// TIA Portal V19 export
FUNCTION "BACKWASH" : Void   // FC13, LAD
{ S7_Optimized_Access := 'TRUE' }
// stored: SetENOAutomatically false
BEGIN

REGION Network 1: BACKWASH_TIMER
END_REGION

REGION Network 2: VALVE OPEN
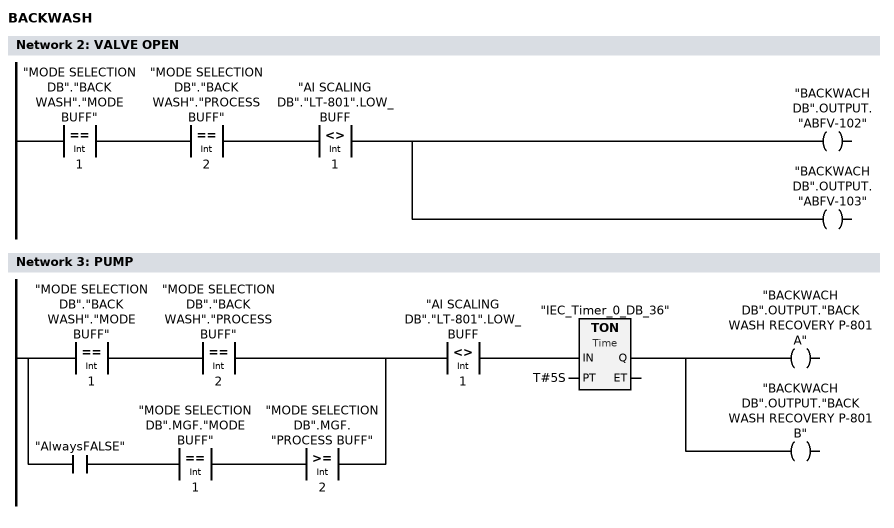
   RUNG wire#powerrail
      { S7_Templates := "SrcType := Int" } EQ_Contact(in1 := "MODE SELECTION DB"."BACK WASH"."MODE BUFF", in2 := 1)
      { S7_Templates := "SrcType := Int" } EQ_Contact(in1 := "MODE SELECTION DB"."BACK WASH"."PROCESS BUFF", in2 := 2)
      { S7_Templates := "SrcType := Int" } NE_Contact(in1 := "AI SCALING DB"."LT-801".LOW_BUFF, in2 := 1)
      wire#w1
      Coil( "BACKWACH DB".OUTPUT."ABFV-102" )
   END_RUNG
   RUNG wire#w1
      Coil( "BACKWACH DB".OUTPUT."ABFV-103" )
   END_RUNG
   // the same network as SCL:
   "BACKWACH DB".OUTPUT."ABFV-102" := ("MODE SELECTION DB"."BACK WASH"."MODE BUFF" = 1) AND ("MODE SELECTION DB"."BACK WASH"."PROCESS BUFF" = 2) AND ("AI SCALING DB"."LT-801".LOW_BUFF <> 1);
   "BACKWACH DB".OUTPUT."ABFV-103" := "BACKWACH DB".OUTPUT."ABFV-102";
END_REGION

REGION Network 3: PUMP
   RUNG wire#powerrail
      { S7_Templates := "SrcType := Int" } EQ_Contact(in1 := "MODE SELECTION DB"."BACK WASH"."MODE BUFF", in2 := 1)
      { S7_Templates := "SrcType := Int" } EQ_Contact(in1 := "MODE SELECTION DB"."BACK WASH"."PROCESS BUFF", in2 := 2)
      wire#w1
      { S7_Templates := "SrcType := Int" } NE_Contact(in1 := "AI SCALING DB"."LT-801".LOW_BUFF, in2 := 1)
      { S7_Templates := "time_type := Time" } "IEC_Timer_0_DB_36".TON(pt := T#5S, et =>)
      wire#w2
      Coil( "BACKWACH DB".OUTPUT."BACK WASH RECOVERY P-801 A" )
   END_RUNG
   RUNG wire#powerrail
      Contact( "AlwaysFALSE" )
      { S7_Templates := "SrcType := Int" } EQ_Contact(in1 := "MODE SELECTION DB".MGF."MODE BUFF", in2 := 1)
      { S7_Templates := "SrcType := Int" } GE_Contact(in1 := "MODE SELECTION DB".MGF."PROCESS BUFF", in2 := 2)
   END_RUNG wire#w1
   RUNG wire#w2
      Coil( "BACKWACH DB".OUTPUT."BACK WASH RECOVERY P-801 B" )
   END_RUNG
   // the same network as SCL:
   "IEC_Timer_0_DB_36".TON(IN := ((("MODE SELECTION DB"."BACK WASH"."MODE BUFF" = 1) AND ("MODE SELECTION DB"."BACK WASH"."PROCESS BUFF" = 2)) OR ("AlwaysFALSE" AND ("MODE SELECTION DB".MGF."MODE BUFF" = 1) AND ("MODE SELECTION DB".MGF."PROCESS BUFF" >= 2))) AND ("AI SCALING DB"."LT-801".LOW_BUFF <> 1),
                           PT := T#5S);
   "BACKWACH DB".OUTPUT."BACK WASH RECOVERY P-801 A" := "IEC_Timer_0_DB_36".Q;
   "BACKWACH DB".OUTPUT."BACK WASH RECOVERY P-801 B" := "IEC_Timer_0_DB_36".Q;
END_REGION
END_FUNCTION
